// TIA Portal project "Lab_01_git" (V16)

(* hardware
DEVICE "S7-1200 station_1"  S7-1200 Station
   slot 0: "Rack_0"  S7-1200 Rack  Rack  V1.0
   slot 1: "PLC_1"  CPU 1214C DC/DC/Rly  6ES7 214-1HG40-0XB0  V4.4
*)

// ===== PLC "PLC_1"  CPU 1214C DC/DC/Rly =====

VAR_GLOBAL   // PLC tag table "Tabla de variables estándar"
   "Tag_1" AT %I0.0 : Bool;
   "Marca2_0" AT %M2.0 : Bool;
   "Tag_2" AT %Q0.0 : Bool;
END_VAR

FUNCTION "Bloque_1" : Void   // FC1, LAD
{ S7_Optimized_Access := 'TRUE' }
VERSION : 0.1
BEGIN
END_FUNCTION

ORGANIZATION_BLOCK "Main"   // OB1, LAD, ProgramCycle
TITLE = "Main Program Sweep (Cycle)"
{ S7_Optimized_Access := 'TRUE' }
VERSION : 0.1
   VAR_INPUT
      Initial_Call : Bool;   // Initial call of this OB
      Remanence : Bool;   // =True, if remanent data are available
   END_VAR
BEGIN

REGION Network 1
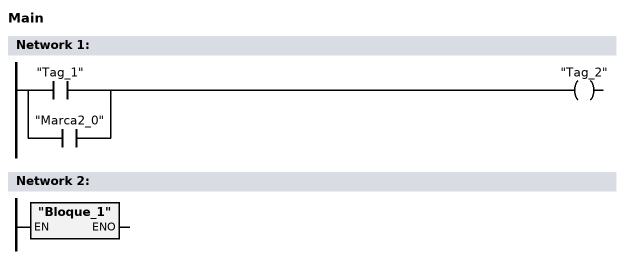
   RUNG wire#powerrail
      Contact( "Tag_1" )
      wire#w1
      Coil( "Tag_2" )
   END_RUNG
   RUNG wire#powerrail
      Contact( "Marca2_0" )
   END_RUNG wire#w1
   // the same network as SCL:
   "Tag_2" := "Tag_1" OR "Marca2_0";
END_REGION

REGION Network 2
   RUNG wire#powerrail
      "Bloque_1"()
   END_RUNG
   // the same network as SCL:
   "Bloque_1"();
END_REGION
END_ORGANIZATION_BLOCK